{attribute addProperty BoxType "ER5151-0002-0018"}
{attribute addProperty Id "ENC_Status_compactAT %I*ENC_Status_compact_3D346E774860ENC_Control_compactAT %Q*ENC_Control_compact_03701F333240WcStateAT %I*WcState_98A4DF7520.250InfoDataAT %I*InfoData_BC63D37F80100"}
{attribute addProperty CRC "2042788864"}
{attribute addProperty SizeInBites "162"}
{attribute addProperty SizeInBytes "20.25"}
TYPE ER5151_19FB32BA :
STRUCT
	{attribute addProperty Name "ENC_Status_compact"}
	ENC_Status_compact : ENC_Status_compact_3D346E77;
	{attribute addProperty Name "ENC_Control_compact"}
	ENC_Control_compact : ENC_Control_compact_03701F33;
	{attribute addProperty Name "WcState"}
	WcState : WcState_98A4DF75;
	{attribute addProperty Name "InfoData"}
	InfoData : InfoData_BC63D37F;
END_STRUCT
END_TYPE

(* stored: Version 1.2.0.0, ProductVersion 3.1.4024.9
   DUT ER5151_19FB32BA: Id {99a6777a-f445-474f-a250-fe7882f363e7} *)
